{attribute 'GeneratedUsingTerminal: EPP7041-1002-0016'}
{attribute addProperty BoxType "EPP7041-1002-0016"}
{attribute addProperty Id "ControlAT %Q*Control_5FD4673D4"}
{attribute addProperty CRC "3125601106"}
{attribute addProperty Size "4"}
TYPE STM_Control_BA4CE352 EXTENDS OutputBase_10CEE7DE :
STRUCT
	{attribute addProperty Name "Control"}
	Control AT %Q* : Control_5FD4673D;
END_STRUCT
END_TYPE

(* stored: Version 1.2.0.0, ProductVersion 3.1.4024.11
   DUT STM_Control_BA4CE352: Id {95d377ad-a55a-4450-b05b-e447dffdf13a} *)
